TYPE UDT_SensorOutput :
STRUCT
	Value: BOOL;
END_STRUCT
END_TYPE

(* stored: Version 1.1.0.1, ProductVersion 3.1.4022.16
   DUT UDT_SensorOutput: Id {d3e1a9ff-cb71-41cd-9498-65ce251de5aa} *)
